Staubli VAL3: checkIoBus.pgx

public program checkIoBus(bool& x_bBool)
  local num l_nStatus
  local num i
begin
  x_bBool=true
  //check bus status
  l_nStatus=ioBusStatus(sIoBusStatus)
  nJishu=size(sIoBusStatus)
  for i=0 to size(sIoBusStatus)-1
    //是否找到了相应的APLICOM端口
    if left(sIoBusStatus[i],1)!="0"
      x_bBool=false
      return
    endIf
  endFor
end
